(* CODESYS project TUT12_PlcLibrary.library
   Company: Beckhoff Automation GmbH
   Title: TUT12_PlcLibrary
   Version: 1.0.0.0

Project tree, tasks and I/O mapping:
  libraries: Tc2_Standard, * (Beckhoff Automation GmbH); Tc2_System, * (Beckhoff Automation GmbH); Tc3_Interfaces, * (Beckhoff Automation GmbH); Tc3_Module, * (Beckhoff Automation GmbH)
  DUTs/
  GVLs/
  POUs/
    program MAIN [ST]
  Version/
    global variables Global_Version
  VISUs/
*)

// Version/Global_Version
// This function has been automatically generated from the project information.
VAR_GLOBAL CONSTANT
	{attribute 'const_non_replaced'}
	stLibVersion_TUT12_PlcLibrary : ST_LibVersion := (iMajor := 1, iMinor := 0, iBuild := 0, iRevision := 0, sVersion := '1.0.0.0');
END_VAR

// POUs/MAIN
PROGRAM MAIN
VAR
	bBool	: BOOL;
END_VAR

bBool := NOT bBool;

END_PROGRAM
